// SIMATIC STEP 7 (V5.x) project TEMA 8 EJERCICIO 6
// CPU: CPU313 C-2 DP(1)
// station: P_ADR_BUS
// station: Hardware
// station: Equipo SIMATIC 300
// program: Programa S7(1)

SYMBOL_TABLE
"FLANCOS"	DB 1	DB 1
"MANIOBRA"	DB 2	DB 2
"MARCHA"	I 0.0	BOOL
"Cycle Execution"	OB 1	OB 1
"S1 VERDE"	Q 0.0	BOOL
"S1 AMBAR"	Q 0.1	BOOL
"S1 ROJO"	Q 0.2	BOOL
"S2 VERDE"	Q 0.3	BOOL
"S2 AMBAR"	Q 0.4	BOOL
"S2 ROJO"	Q 0.5	BOOL
"VAT_1"	VAT 1	
END_SYMBOL_TABLE

DATA_BLOCK "FLANCOS"	// DB 1
VERSION : 0.1
  STRUCT
   MARCA0 : BOOL ;
   MARCA1 : BOOL ;
   MARCA2 : BOOL ;
   MARCA3 : BOOL ;
   MARCA4 : BOOL ;
   MARCA5 : BOOL ;
   MARCA6 : BOOL ;
   MARCA7 : BOOL ;
   MARCA10 : BOOL ;
   MARCA11 : BOOL ;
   MARCA12 : BOOL ;
   MARCA13 : BOOL ;
   MARCA14 : BOOL ;
   MARCA15 : BOOL ;
   MARCA16 : BOOL ;
   MARCA17 : BOOL ;
   MARCA20 : BOOL ;
   MARCA21 : BOOL ;
   MARCA22 : BOOL ;
   MARCA23 : BOOL ;
   MARCA24 : BOOL ;
   MARCA25 : BOOL ;
   MARCA26 : BOOL ;
   MARCA27 : BOOL ;
  END_STRUCT ;	
BEGIN
END_DATA_BLOCK

DATA_BLOCK "MANIOBRA"	// DB 2
VERSION : 0.1
  STRUCT
   M0 : BOOL ;
   M1 : BOOL ;
   M2 : BOOL ;
   M3 : BOOL ;
   M4 : BOOL ;
   M5 : BOOL ;
   M6 : BOOL ;
   M7 : BOOL ;
   M10 : BOOL ;
   M11 : BOOL ;
   M12 : BOOL ;
   M13 : BOOL ;
  END_STRUCT ;	
BEGIN
END_DATA_BLOCK

ORGANIZATION_BLOCK "Cycle Execution"	// OB 1
TITLE = "Main Program Sweep (Cycle)"
//CRUCE REGULADO POR 2 SEMAFOROS PARA COCHES CON SECUENCIAS TEMPORIZADAS 
//INDEPENDIENTES
VERSION : 0.1
VAR_TEMP
  OB1_EV_CLASS : BYTE ;	//Bits 0-3 = 1 (Coming event), Bits 4-7 = 1 (Event class 1)
  OB1_SCAN_1 : BYTE ;	//1 (Cold restart scan 1 of OB 1), 3 (Scan 2-n of OB 1)
  OB1_PRIORITY : BYTE ;	//Priority of OB Execution
  OB1_OB_NUMBR : BYTE ;	//1 (Organization block 1, OB1)
  OB1_RESERVED_1 : BYTE ;	//Reserved for system
  OB1_RESERVED_2 : BYTE ;	//Reserved for system
  OB1_PREV_CYCLE : INT ;	//Cycle time of previous OB1 scan (milliseconds)
  OB1_MIN_CYCLE : INT ;	//Minimum cycle time of OB1 (milliseconds)
  OB1_MAX_CYCLE : INT ;	//Maximum cycle time of OB1 (milliseconds)
  OB1_DATE_TIME : DATE_AND_TIME ;	//Date and time OB1 started
END_VAR
BEGIN
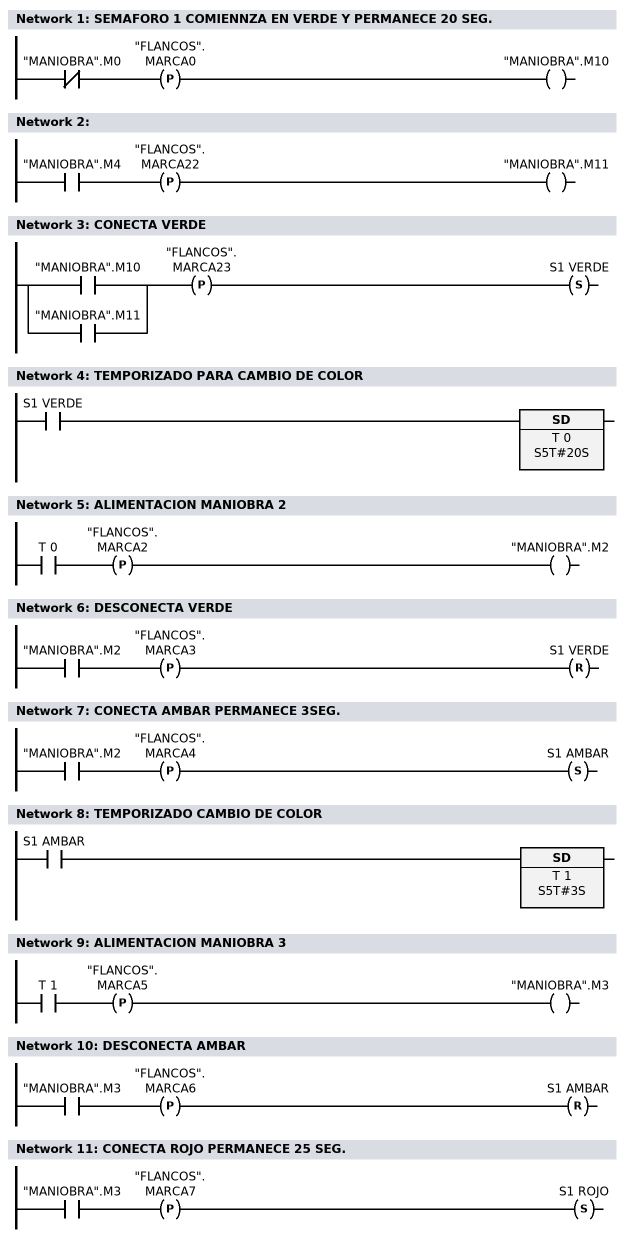
NETWORK
TITLE = SEMAFORO 1 COMIENNZA EN VERDE Y PERMANECE 20 SEG. 
//CONTACTO CERRADO DE MANIOBRA 0 MANDA UN PULSO EN EL PRIMER CICLO PARA EMPEZAR 
//LA 
//SECUENCIA 
      AN    "MANIOBRA".M0;
      FP    "FLANCOS".MARCA0;
      =     "MANIOBRA".M10;
NETWORK
TITLE =
//MANIOBRA 4 ENVIA UN PULSO PARA QUE FUNCIONE PERMANENTE DE FORMA CICLICA
      A     "MANIOBRA".M4;
      FP    "FLANCOS".MARCA22;
      =     "MANIOBRA".M11;
NETWORK
TITLE = CONECTA VERDE 
      A(;
      O     "MANIOBRA".M10;
      O     "MANIOBRA".M11;
      );
      FP    "FLANCOS".MARCA23;
      S     "S1 VERDE";
NETWORK
TITLE = TEMPORIZADO PARA CAMBIO DE COLOR
//T0 SE 20 SEG.
      A     "S1 VERDE";
      L     S5T#20S;
      SD    T 0;
NETWORK
TITLE = ALIMENTACION MANIOBRA 2
      A     T 0;
      FP    "FLANCOS".MARCA2;
      =     "MANIOBRA".M2;
NETWORK
TITLE = DESCONECTA VERDE 
      A     "MANIOBRA".M2;
      FP    "FLANCOS".MARCA3;
      R     "S1 VERDE";
NETWORK
TITLE = CONECTA AMBAR PERMANECE 3SEG.
      A     "MANIOBRA".M2;
      FP    "FLANCOS".MARCA4;
      S     "S1 AMBAR";
NETWORK
TITLE = TEMPORIZADO CAMBIO DE COLOR
//T1 SE 3 SEG.
      A     "S1 AMBAR";
      L     S5T#3S;
      SD    T 1;
NETWORK
TITLE = ALIMENTACION MANIOBRA 3
      A     T 1;
      FP    "FLANCOS".MARCA5;
      =     "MANIOBRA".M3;
NETWORK
TITLE = DESCONECTA AMBAR
      A     "MANIOBRA".M3;
      FP    "FLANCOS".MARCA6;
      R     "S1 AMBAR";
NETWORK
TITLE = CONECTA ROJO PERMANECE 25 SEG.
      A     "MANIOBRA".M3;
      FP    "FLANCOS".MARCA7;
      S     "S1 ROJO";
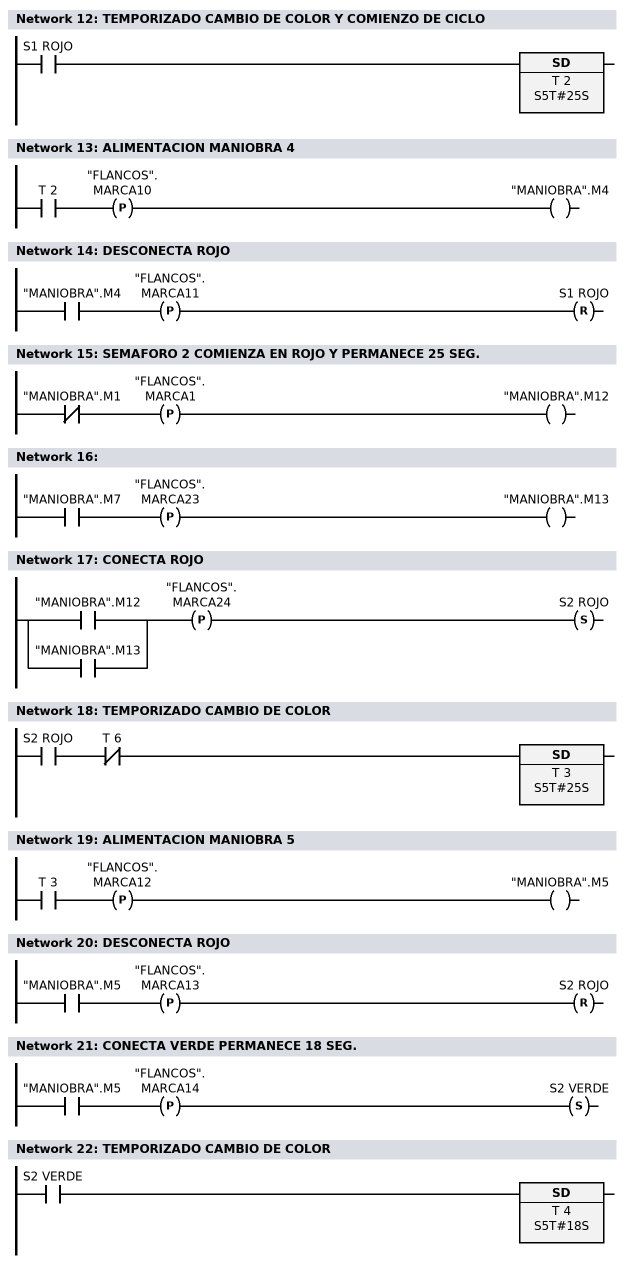
NETWORK
TITLE = TEMPORIZADO CAMBIO DE COLOR Y COMIENZO DE CICLO
//T2 SE 25  SEG.
      A     "S1 ROJO";
      L     S5T#25S;
      SD    T 2;
NETWORK
TITLE = ALIMENTACION MANIOBRA 4
      A     T 2;
      FP    "FLANCOS".MARCA10;
      =     "MANIOBRA".M4;
NETWORK
TITLE = DESCONECTA ROJO
//MANIOBRA 4 SERA LA ENCARGADA DE ENVIAR UN PULSO PARA INICIAR LA SECUENCIA DE 
//FORMA CICLICA
      A     "MANIOBRA".M4;
      FP    "FLANCOS".MARCA11;
      R     "S1 ROJO";
NETWORK
TITLE = SEMAFORO 2 COMIENZA EN ROJO Y PERMANECE 25 SEG.
// CONTACTO CERRADA ENVIA UN PULSO EN EL PRIMER CICLO PARA EMPEZAR LA SECUENCIA
      AN    "MANIOBRA".M1;
      FP    "FLANCOS".MARCA1;
      =     "MANIOBRA".M12;
NETWORK
TITLE =
//MANIOBRA ENVIA UN PULSO PARA QUE FUNCIONE DE FORMA PERMANENTE CICLICA
      A     "MANIOBRA".M7;
      FP    "FLANCOS".MARCA23;
      =     "MANIOBRA".M13;
NETWORK
TITLE = CONECTA ROJO
      A(;
      O     "MANIOBRA".M12;
      O     "MANIOBRA".M13;
      );
      FP    "FLANCOS".MARCA24;
      S     "S2 ROJO";
NETWORK
TITLE = TEMPORIZADO CAMBIO DE COLOR
//T3 SE 25 SEG.
      A     "S2 ROJO";
      AN    T 6;
      L     S5T#25S;
      SD    T 3;
NETWORK
TITLE = ALIMENTACION MANIOBRA 5
      A     T 3;
      FP    "FLANCOS".MARCA12;
      =     "MANIOBRA".M5;
NETWORK
TITLE = DESCONECTA ROJO
      A     "MANIOBRA".M5;
      FP    "FLANCOS".MARCA13;
      R     "S2 ROJO";
NETWORK
TITLE = CONECTA VERDE PERMANECE 18 SEG.
      A     "MANIOBRA".M5;
      FP    "FLANCOS".MARCA14;
      S     "S2 VERDE";
NETWORK
TITLE = TEMPORIZADO CAMBIO DE COLOR
//T4 SE 18 SEG.
      A     "S2 VERDE";
      L     S5T#18S;
      SD    T 4;
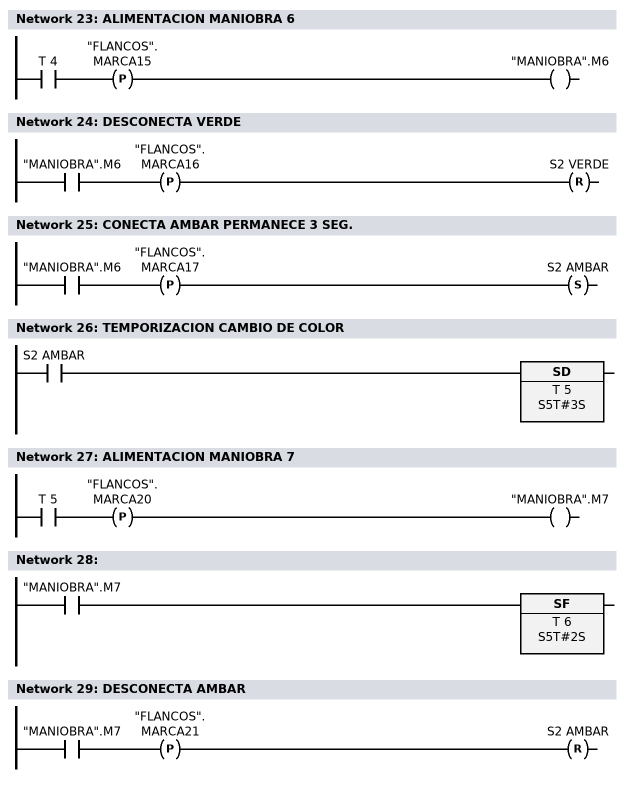
NETWORK
TITLE = ALIMENTACION MANIOBRA 6
      A     T 4;
      FP    "FLANCOS".MARCA15;
      =     "MANIOBRA".M6;
NETWORK
TITLE = DESCONECTA VERDE
      A     "MANIOBRA".M6;
      FP    "FLANCOS".MARCA16;
      R     "S2 VERDE";
NETWORK
TITLE = CONECTA AMBAR PERMANECE 3 SEG.
      A     "MANIOBRA".M6;
      FP    "FLANCOS".MARCA17;
      S     "S2 AMBAR";
NETWORK
TITLE = TEMPORIZACION CAMBIO DE COLOR 
//T5 SE 3 SEG.
      A     "S2 AMBAR";
      L     S5T#3S;
      SD    T 5;
NETWORK
TITLE = ALIMENTACION MANIOBRA 7
//MANIOBRA 7 ES LA ENCARGADA DE ENVIAR UN PULSO PARA VOLVER A INICIAR LA 
//SECUENCIA 
//DE FORMA CICLICA
      A     T 5;
      FP    "FLANCOS".MARCA20;
      =     "MANIOBRA".M7;
NETWORK
TITLE =
      A     "MANIOBRA".M7;
      L     S5T#2S;
      SF    T 6;
NETWORK
TITLE = DESCONECTA AMBAR 
      A     "MANIOBRA".M7;
      FP    "FLANCOS".MARCA21;
      R     "S2 AMBAR";
END_ORGANIZATION_BLOCK
